INTERFACE I_WashStrategy

METHOD GetDuration : TIME
END_METHOD

METHOD Start 
VAR_IN_OUT
    config : ST_MachineConfig;
END_VAR
END_METHOD

END_INTERFACE

(* stored: Version 1.1.0.1, ProductVersion 3.1.4024.16
   Itf I_WashStrategy: Id {5fa598a7-78ea-4ca8-9727-001f86b81944}
   Method GetDuration: Id {4c64d98c-0676-4393-93d4-a58eb978ce16}
   Method Start: Id {de175e78-f862-4276-9927-97214fdaa317} *)
